TYPE stHMI_SKILL :
STRUCT
	bExecute : BOOL;
    bStop    : BOOL;
	Tag		: STRING;
// 	{attribute 'OPC.UA.DA.StructuredType':=1}		//TODO
// 	{attribute 'OPC.UA.DA' := '1'}
//     Status    : stExternalStatus;
// 	{attribute 'OPC.UA.DA.StructuredType':=1}
// 	{attribute 'OPC.UA.DA' := '1'}
//     Command   : stExternalCommand;
END_STRUCT
END_TYPE

(* stored: Version 1.1.0.1, ProductVersion 3.1.4026.18
   DUT stHMI_SKILL: Id {a747dac1-4524-4a05-be3b-8256e4b5a769} *)
